(* Logix 5000 project; controller PRU vendor 1 type 14 code 107 rev 20.13; software revision 20.01; part 13 of 17 *)
(* tags used below, declared in another part *)
   AI0_CALCULATED : REAL;
   AI0_WF : DSi_WF50;
   AI10_CALCULATED : REAL;
   AI10_WF : DSi_WF50;
   AI11_CALCULATED : REAL;
   AI11_WF : DSi_WF50;
   AI12_CALCULATED : REAL;
   AI12_WF : DSi_WF50;
   AI13_CALCULATED : REAL;
   AI13_WF : DSi_WF50;
   AI14_CALCULATED : REAL;
   AI14_WF : DSi_WF50;
   AI15_CALCULATED : REAL;
   AI15_WF : DSi_WF50;
   AI16_CALCULATED : REAL;
   AI16_WF : DSi_WF50;
   AI1_CALCULATED : REAL;
   AI1_WF : DSi_WF50;
   AI2_CALCULATED : REAL;
   AI2_WF : DSi_WF50;
   AI3_CALCULATED : REAL;
   AI3_WF : DSi_WF50;
   AI4_CALCULATED : REAL;
   AI4_WF : DSi_WF50;
   AI5_CALCULATED : REAL;
   AI5_WF : DSi_WF50;
   AI6_CALCULATED : REAL;
   AI6_WF : DSi_WF50;
   AI7_CALCULATED : REAL;
   AI7_WF : DSi_WF50;
   AI8_CALCULATED : REAL;
   AI8_WF : DSi_WF50;
   AI9_CALCULATED : REAL;
   AI9_WF : DSi_WF50;
   AI_0 : AI_1769_IF4;
   AI_0_FILTERED : DINT;
   AI_1 : AI_1769_IF4;
   AI_10 : AI_1769_IF4;
   AI_10_FILTERED : REAL;
   AI_11 : AI_1769_IF4;
   AI_11_FILTERED : REAL;
   AI_12 : AI_1769_IF4;
   AI_12_FILTERED : REAL;
   AI_13 : AI_1769_IF4;
   AI_13_FILTERED : REAL;
   AI_14 : AI_1769_IF4;
   AI_14_FILTERED : REAL;
   AI_15 : AI_1769_IF4;
   AI_15_FILTERED : REAL;
   AI_16 : AI_1769_IF4;
   AI_16_DATA : REAL;
   AI_16_FILTERED : REAL;
   AI_1_FILTERED : REAL;
   AI_2 : AI_1769_IF4;
   AI_2_FILTERED : REAL;
   AI_3 : AI_1769_IF4;
   AI_3_FILTERED : REAL;
   AI_4 : AI_1769_IF4;
   AI_4_FILTERED : REAL;
   AI_5 : AI_1769_IF4;
   AI_5_FILTERED : REAL;
   AI_6 : AI_1769_IF4;
   AI_6_FILTERED : REAL;
   AI_7 : AI_1769_IF4;
   AI_7_FILTERED : REAL;
   AI_8 : AI_1769_IF4;
   AI_8_FILTERED : REAL;
   AI_9 : AI_1769_IF4;
   AI_9_FILTERED : REAL;
   CALC_SPARE_AO_CMD : REAL;
   CSS_CommsLoss_TMR : TIMER;
   CSS_CommsLossAlm : BOOL;
   CSS_CommsWarning_TMR : TIMER;
   CSS_CommsWarningAlm : BOOL;
   CSS_PLC_Seconds_Temp : DINT;
   CSS_Status_Data : PLCStatusData;
   DisableAllHeaters : BOOL;
   HMI_Ai0_FORCE : BOOL;
   HMI_Ai0_FORCE_VALUE : REAL;
   HMI_AI0_HI_SCALE : REAL;
   HMI_AI0_LO_SCALE : REAL;
   HMI_Ai10_FORCE : BOOL;
   HMI_Ai10_FORCE_VALUE : REAL;
   HMI_AI10_HI_SCALE : REAL;
   HMI_AI10_LO_SCALE : REAL;
   HMI_Ai11_FORCE : BOOL;
   HMI_Ai11_FORCE_VALUE : REAL;
   HMI_AI11_HI_SCALE : REAL;
   HMI_AI11_LO_SCALE : REAL;
   HMI_Ai12_FORCE : BOOL;
   HMI_Ai12_FORCE_VALUE : REAL;
   HMI_AI12_HI_SCALE : REAL;
   HMI_AI12_LO_SCALE : REAL;
   HMI_Ai13_FORCE : BOOL;
   HMI_Ai13_FORCE_VALUE : REAL;
   HMI_AI13_HI_SCALE : REAL;
   HMI_AI13_LO_SCALE : REAL;
   HMI_Ai14_FORCE : BOOL;
   HMI_Ai14_FORCE_VALUE : REAL;
   HMI_AI14_HI_SCALE : REAL;
   HMI_AI14_LO_SCALE : REAL;
   HMI_Ai15_FORCE : BOOL;
   HMI_Ai15_FORCE_VALUE : REAL;
   HMI_AI15_HI_SCALE : REAL;
   HMI_AI15_LO_SCALE : REAL;
   HMI_AI16_FORCE : BOOL;
   HMI_AI16_FORCE_VALUE : REAL;
   HMI_AI16_HI_SCALE : REAL;
   HMI_AI16_LO_SCALE : REAL;
   HMI_Ai1_FORCE : BOOL;
   HMI_Ai1_FORCE_VALUE : REAL;
   HMI_AI1_HI_SCALE : REAL;
   HMI_AI1_LO_SCALE : REAL;
   HMI_Ai2_FORCE : BOOL;
   HMI_Ai2_FORCE_VALUE : REAL;
   HMI_AI2_HI_SCALE : REAL;
   HMI_AI2_LO_SCALE : REAL;
   HMI_Ai3_FORCE : BOOL;
   HMI_Ai3_FORCE_VALUE : REAL;
   HMI_AI3_HI_SCALE : REAL;
   HMI_AI3_LO_SCALE : REAL;
   HMI_Ai4_FORCE : BOOL;
   HMI_Ai4_FORCE_VALUE : REAL;
   HMI_AI4_HI_SCALE : REAL;
   HMI_AI4_LO_SCALE : REAL;
   HMI_Ai5_FORCE : BOOL;
   HMI_Ai5_FORCE_VALUE : REAL;
   HMI_AI5_HI_SCALE : REAL;
   HMI_AI5_LO_SCALE : REAL;
   HMI_Ai6_FORCE : BOOL;
   HMI_Ai6_FORCE_VALUE : REAL;
   HMI_AI6_HI_SCALE : REAL;
   HMI_AI6_LO_SCALE : REAL;
   HMI_Ai7_FORCE : BOOL;
   HMI_Ai7_FORCE_VALUE : REAL;
   HMI_AI7_HI_SCALE : REAL;
   HMI_AI7_LO_SCALE : REAL;
   HMI_Ai8_FORCE : BOOL;
   HMI_Ai8_FORCE_VALUE : REAL;
   HMI_AI8_HI_SCALE : REAL;
   HMI_AI8_LO_SCALE : REAL;
   HMI_Ai9_FORCE : BOOL;
   HMI_Ai9_FORCE_VALUE : REAL;
   HMI_AI9_HI_SCALE : REAL;
   HMI_AI9_LO_SCALE : REAL;
   HMI_HTR1_FORCED : BOOL;
   HMI_HTR1_POWER_CMD : REAL;
   HMI_HTR2_FORCED : BOOL;
   HMI_HTR2_POWER_CMD : REAL;
   HMI_HTR3_FORCED : BOOL;
   HMI_HTR3_POWER_CMD : REAL;
   HMI_HTR4_FORCED : BOOL;
   HMI_HTR4_POWER_CMD : REAL;
   HMI_HTR5_FORCED : BOOL;
   HMI_HTR5_POWER_CMD : REAL;
   HMI_HTR6_FORCED : BOOL;
   HMI_HTR6_POWER_CMD : REAL;
   HMI_HTR7_FORCED : BOOL;
   HMI_HTR7_POWER_CMD : REAL;
   HMI_HTR8_FORCED : BOOL;
   HMI_HTR8_POWER_CMD : REAL;
   HMI_HTR9_FORCED : BOOL;
   HMI_HTR9_POWER_CMD : REAL;
   HMI_SPARE_AO_CMD : REAL;
   HMI_SPARE_AO_FORCED : BOOL;
   HTR1_POWER_CMD : REAL;
   HTR2_POWER_CMD : REAL;
   HTR3_POWER_CMD : REAL;
   HTR4_POWER_CMD : REAL;
   HTR5_POWER_CMD : REAL;
   HTR6_POWER_CMD : REAL;
   HTR7_POWER_CMD : REAL;
   HTR8_POWER_CMD : REAL;
   HTR9_POWER_CMD : REAL;
   Major : DINT;
   Minor : DINT;
   Revision : DINT;
   SPARE_AO_CMD : REAL;
   TOTE_WEIGHT : REAL;
   UTL_Status_Data : PLCStatusData;
   Z1_AMPS_TEMP : REAL;
   Z1_L1_AMPS : REAL;
   Z1_L2_AMPS : REAL;
   Z1_L3_AMPS : REAL;
   Z1L1_Tot : EnergyTot;
   Z1L2_Tot : EnergyTot;
   Z1L3_Tot : EnergyTot;
   Z2_AMPS_TEMP : REAL;
   Z2_L1_AMPS : REAL;
   Z2_L2_AMPS : REAL;
   Z2_L3_AMPS : REAL;
   Z2L1_Tot : EnergyTot;
   Z2L2_Tot : EnergyTot;
   Z2L3_Tot : EnergyTot;
   Z3_AMPS_TEMP : REAL;
   Z3_L1_AMPS : REAL;
   Z3_L2_AMPS : REAL;
   Z3_L3_AMPS : REAL;
   Z3L1_Tot : EnergyTot;
   Z3L2_Tot : EnergyTot;
   Z3L3_Tot : EnergyTot;
   Z4_L1_AMPS : REAL;
   Z4L1_Tot : EnergyTot;
   Z5_L2_AMPS : REAL;
   Z5L2_Tot : EnergyTot;
   Z6_L3_AMPS : REAL;
   Z6L3_Tot : EnergyTot;
   Z7_L1_AMPS : REAL;
   Z7L1_Tot : EnergyTot;
   Z8_L2_AMPS : REAL;
   Z8L2_Tot : EnergyTot;
   Z9_L3_AMPS : REAL;
   Z9L3_Tot : EnergyTot;
   ZONE_1_AMPS : DINT;
   ZONE_1_POWER_CMD : REAL;
   ZONE_2_AMPS : DINT;
   ZONE_2_POWER_CMD : REAL;
   ZONE_3_AMPS : DINT;
   ZONE_3_POWER_CMD : REAL;
   ZONE_4_AMPS : DINT;
   ZONE_4_POWER_CMD : REAL;
   ZONE_5_AMPS : DINT;
   ZONE_5_POWER_CMD : REAL;
   ZONE_6_AMPS : DINT;
   ZONE_6_POWER_CMD : REAL;
   ZONE_7_AMPS : DINT;
   ZONE_7_POWER_CMD : REAL;
   ZONE_8_AMPS : DINT;
   ZONE_8_POWER_CMD : REAL;
   ZONE_9_AMPS : DINT;
   ZONE_9_POWER_CMD : REAL;
(* MainProgram, continued *)

ROUTINE G04_MAP_ANALOG_INPUTS   (* ladder *)
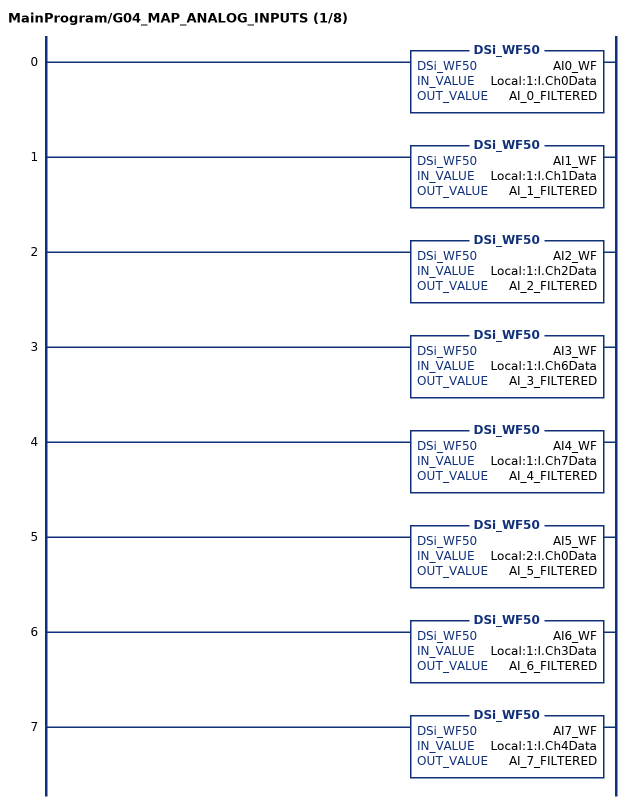
   0: DSi_WF50(AI0_WF,Local:1:I.Ch0Data,AI_0_FILTERED);
   1: DSi_WF50(AI1_WF,Local:1:I.Ch1Data,AI_1_FILTERED);
   2: DSi_WF50(AI2_WF,Local:1:I.Ch2Data,AI_2_FILTERED);
   3: DSi_WF50(AI3_WF,Local:1:I.Ch6Data,AI_3_FILTERED);
   4: DSi_WF50(AI4_WF,Local:1:I.Ch7Data,AI_4_FILTERED);
   5: DSi_WF50(AI5_WF,Local:2:I.Ch0Data,AI_5_FILTERED);
   6: DSi_WF50(AI6_WF,Local:1:I.Ch3Data,AI_6_FILTERED);
   7: DSi_WF50(AI7_WF,Local:1:I.Ch4Data,AI_7_FILTERED);
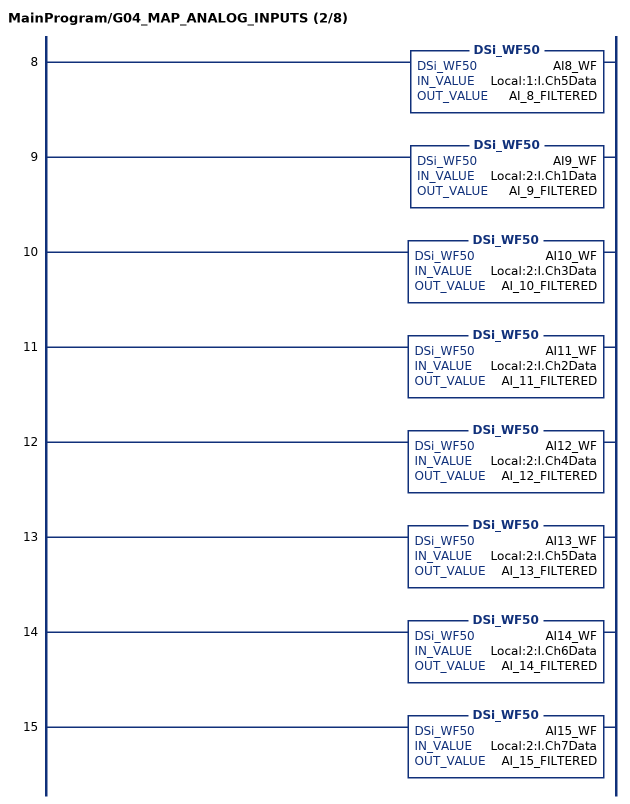
   8: DSi_WF50(AI8_WF,Local:1:I.Ch5Data,AI_8_FILTERED);
   9: DSi_WF50(AI9_WF,Local:2:I.Ch1Data,AI_9_FILTERED);
   10: DSi_WF50(AI10_WF,Local:2:I.Ch3Data,AI_10_FILTERED);
   11: DSi_WF50(AI11_WF,Local:2:I.Ch2Data,AI_11_FILTERED);
   12: DSi_WF50(AI12_WF,Local:2:I.Ch4Data,AI_12_FILTERED);
   13: DSi_WF50(AI13_WF,Local:2:I.Ch5Data,AI_13_FILTERED);
   14: DSi_WF50(AI14_WF,Local:2:I.Ch6Data,AI_14_FILTERED);
   15: DSi_WF50(AI15_WF,Local:2:I.Ch7Data,AI_15_FILTERED);
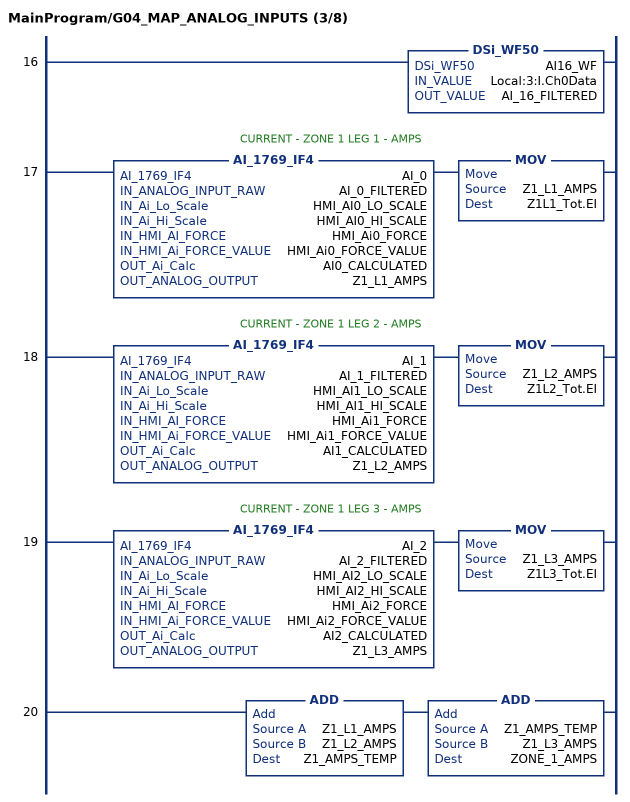
   16: DSi_WF50(AI16_WF,Local:3:I.Ch0Data,AI_16_FILTERED);
   // CURRENT - ZONE 1 LEG 1 - AMPS
   17: AI_1769_IF4(AI_0,AI_0_FILTERED,HMI_AI0_LO_SCALE,HMI_AI0_HI_SCALE,HMI_Ai0_FORCE,HMI_Ai0_FORCE_VALUE,AI0_CALCULATED,Z1_L1_AMPS)MOV(Z1_L1_AMPS,Z1L1_Tot.EI);
   // CURRENT - ZONE 1 LEG 2 - AMPS
   18: AI_1769_IF4(AI_1,AI_1_FILTERED,HMI_AI1_LO_SCALE,HMI_AI1_HI_SCALE,HMI_Ai1_FORCE,HMI_Ai1_FORCE_VALUE,AI1_CALCULATED,Z1_L2_AMPS)MOV(Z1_L2_AMPS,Z1L2_Tot.EI);
   // CURRENT - ZONE 1 LEG 3 - AMPS
   19: AI_1769_IF4(AI_2,AI_2_FILTERED,HMI_AI2_LO_SCALE,HMI_AI2_HI_SCALE,HMI_Ai2_FORCE,HMI_Ai2_FORCE_VALUE,AI2_CALCULATED,Z1_L3_AMPS)MOV(Z1_L3_AMPS,Z1L3_Tot.EI);
   20: ADD(Z1_L1_AMPS,Z1_L2_AMPS,Z1_AMPS_TEMP)ADD(Z1_AMPS_TEMP,Z1_L3_AMPS,ZONE_1_AMPS);
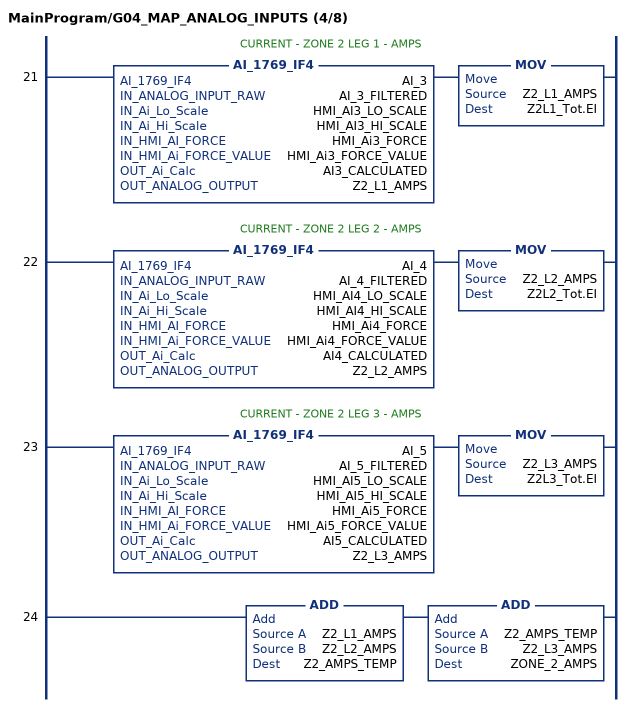
   // CURRENT - ZONE 2 LEG 1 - AMPS
   21: AI_1769_IF4(AI_3,AI_3_FILTERED,HMI_AI3_LO_SCALE,HMI_AI3_HI_SCALE,HMI_Ai3_FORCE,HMI_Ai3_FORCE_VALUE,AI3_CALCULATED,Z2_L1_AMPS)MOV(Z2_L1_AMPS,Z2L1_Tot.EI);
   // CURRENT - ZONE 2 LEG 2 - AMPS
   22: AI_1769_IF4(AI_4,AI_4_FILTERED,HMI_AI4_LO_SCALE,HMI_AI4_HI_SCALE,HMI_Ai4_FORCE,HMI_Ai4_FORCE_VALUE,AI4_CALCULATED,Z2_L2_AMPS)MOV(Z2_L2_AMPS,Z2L2_Tot.EI);
   // CURRENT - ZONE 2 LEG 3 - AMPS
   23: AI_1769_IF4(AI_5,AI_5_FILTERED,HMI_AI5_LO_SCALE,HMI_AI5_HI_SCALE,HMI_Ai5_FORCE,HMI_Ai5_FORCE_VALUE,AI5_CALCULATED,Z2_L3_AMPS)MOV(Z2_L3_AMPS,Z2L3_Tot.EI);
   24: ADD(Z2_L1_AMPS,Z2_L2_AMPS,Z2_AMPS_TEMP)ADD(Z2_AMPS_TEMP,Z2_L3_AMPS,ZONE_2_AMPS);
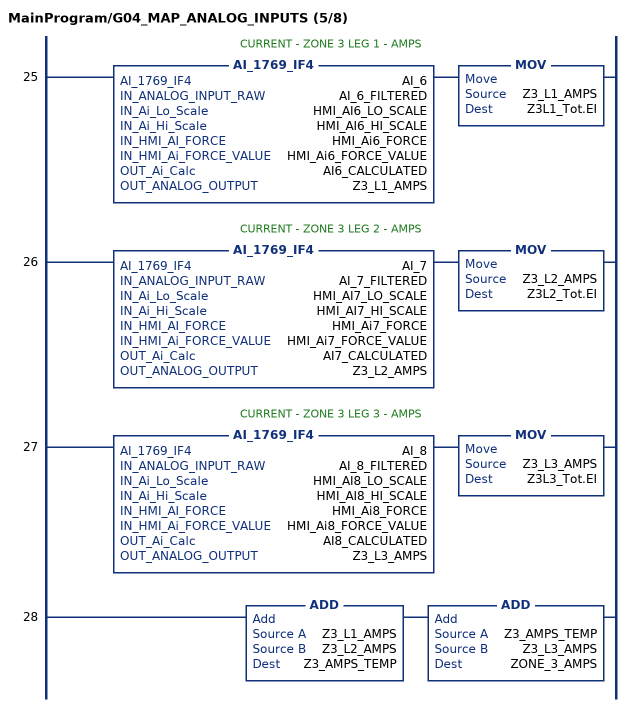
   // CURRENT - ZONE 3 LEG 1 - AMPS
   25: AI_1769_IF4(AI_6,AI_6_FILTERED,HMI_AI6_LO_SCALE,HMI_AI6_HI_SCALE,HMI_Ai6_FORCE,HMI_Ai6_FORCE_VALUE,AI6_CALCULATED,Z3_L1_AMPS)MOV(Z3_L1_AMPS,Z3L1_Tot.EI);
   // CURRENT - ZONE 3 LEG 2 - AMPS
   26: AI_1769_IF4(AI_7,AI_7_FILTERED,HMI_AI7_LO_SCALE,HMI_AI7_HI_SCALE,HMI_Ai7_FORCE,HMI_Ai7_FORCE_VALUE,AI7_CALCULATED,Z3_L2_AMPS)MOV(Z3_L2_AMPS,Z3L2_Tot.EI);
   // CURRENT - ZONE 3 LEG 3 - AMPS
   27: AI_1769_IF4(AI_8,AI_8_FILTERED,HMI_AI8_LO_SCALE,HMI_AI8_HI_SCALE,HMI_Ai8_FORCE,HMI_Ai8_FORCE_VALUE,AI8_CALCULATED,Z3_L3_AMPS)MOV(Z3_L3_AMPS,Z3L3_Tot.EI);
   28: ADD(Z3_L1_AMPS,Z3_L2_AMPS,Z3_AMPS_TEMP)ADD(Z3_AMPS_TEMP,Z3_L3_AMPS,ZONE_3_AMPS);
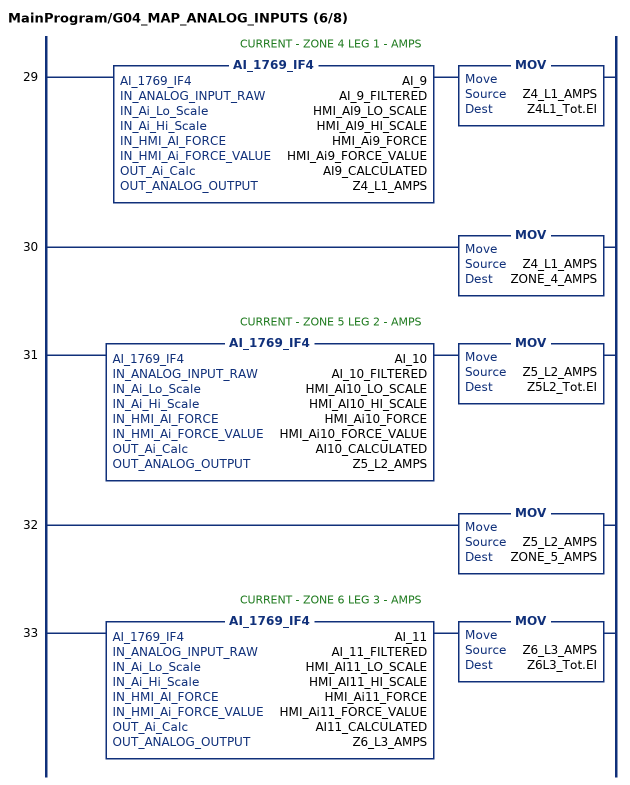
   // CURRENT - ZONE 4 LEG 1 - AMPS
   29: AI_1769_IF4(AI_9,AI_9_FILTERED,HMI_AI9_LO_SCALE,HMI_AI9_HI_SCALE,HMI_Ai9_FORCE,HMI_Ai9_FORCE_VALUE,AI9_CALCULATED,Z4_L1_AMPS)MOV(Z4_L1_AMPS,Z4L1_Tot.EI);
   30: MOV(Z4_L1_AMPS,ZONE_4_AMPS);
   // CURRENT - ZONE 5 LEG 2 - AMPS
   31: AI_1769_IF4(AI_10,AI_10_FILTERED,HMI_AI10_LO_SCALE,HMI_AI10_HI_SCALE,HMI_Ai10_FORCE,HMI_Ai10_FORCE_VALUE,AI10_CALCULATED,Z5_L2_AMPS)MOV(Z5_L2_AMPS,Z5L2_Tot.EI);
   32: MOV(Z5_L2_AMPS,ZONE_5_AMPS);
   // CURRENT - ZONE 6 LEG 3 - AMPS
   33: AI_1769_IF4(AI_11,AI_11_FILTERED,HMI_AI11_LO_SCALE,HMI_AI11_HI_SCALE,HMI_Ai11_FORCE,HMI_Ai11_FORCE_VALUE,AI11_CALCULATED,Z6_L3_AMPS)MOV(Z6_L3_AMPS,Z6L3_Tot.EI);
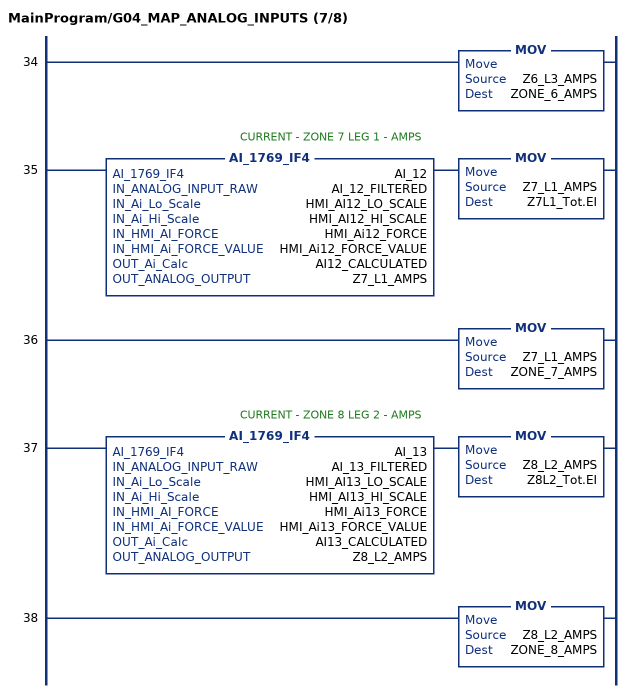
   34: MOV(Z6_L3_AMPS,ZONE_6_AMPS);
   // CURRENT - ZONE 7 LEG 1 - AMPS
   35: AI_1769_IF4(AI_12,AI_12_FILTERED,HMI_AI12_LO_SCALE,HMI_AI12_HI_SCALE,HMI_Ai12_FORCE,HMI_Ai12_FORCE_VALUE,AI12_CALCULATED,Z7_L1_AMPS)MOV(Z7_L1_AMPS,Z7L1_Tot.EI);
   36: MOV(Z7_L1_AMPS,ZONE_7_AMPS);
   // CURRENT - ZONE 8 LEG 2 - AMPS
   37: AI_1769_IF4(AI_13,AI_13_FILTERED,HMI_AI13_LO_SCALE,HMI_AI13_HI_SCALE,HMI_Ai13_FORCE,HMI_Ai13_FORCE_VALUE,AI13_CALCULATED,Z8_L2_AMPS)MOV(Z8_L2_AMPS,Z8L2_Tot.EI);
   38: MOV(Z8_L2_AMPS,ZONE_8_AMPS);
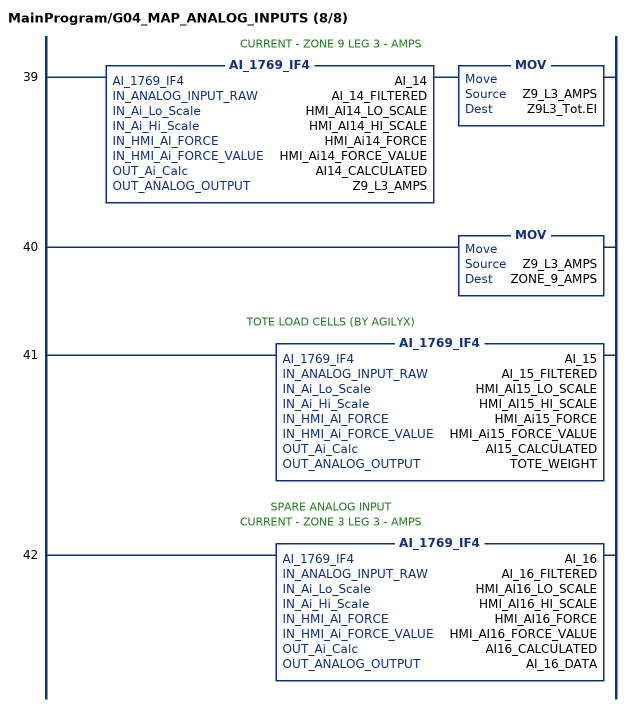
   // CURRENT - ZONE 9 LEG 3 - AMPS
   39: AI_1769_IF4(AI_14,AI_14_FILTERED,HMI_AI14_LO_SCALE,HMI_AI14_HI_SCALE,HMI_Ai14_FORCE,HMI_Ai14_FORCE_VALUE,AI14_CALCULATED,Z9_L3_AMPS)MOV(Z9_L3_AMPS,Z9L3_Tot.EI);
   40: MOV(Z9_L3_AMPS,ZONE_9_AMPS);
   // TOTE LOAD CELLS (BY AGILYX)
   41: AI_1769_IF4(AI_15,AI_15_FILTERED,HMI_AI15_LO_SCALE,HMI_AI15_HI_SCALE,HMI_Ai15_FORCE,HMI_Ai15_FORCE_VALUE,AI15_CALCULATED,TOTE_WEIGHT);
   // SPARE ANALOG INPUT
   // CURRENT - ZONE 3 LEG 3 - AMPS
   42: AI_1769_IF4(AI_16,AI_16_FILTERED,HMI_AI16_LO_SCALE,HMI_AI16_HI_SCALE,HMI_AI16_FORCE,HMI_AI16_FORCE_VALUE,AI16_CALCULATED,AI_16_DATA);
END_ROUTINE

ROUTINE G05_MAP_ANALOG_OUTPUTS   (* ladder *)
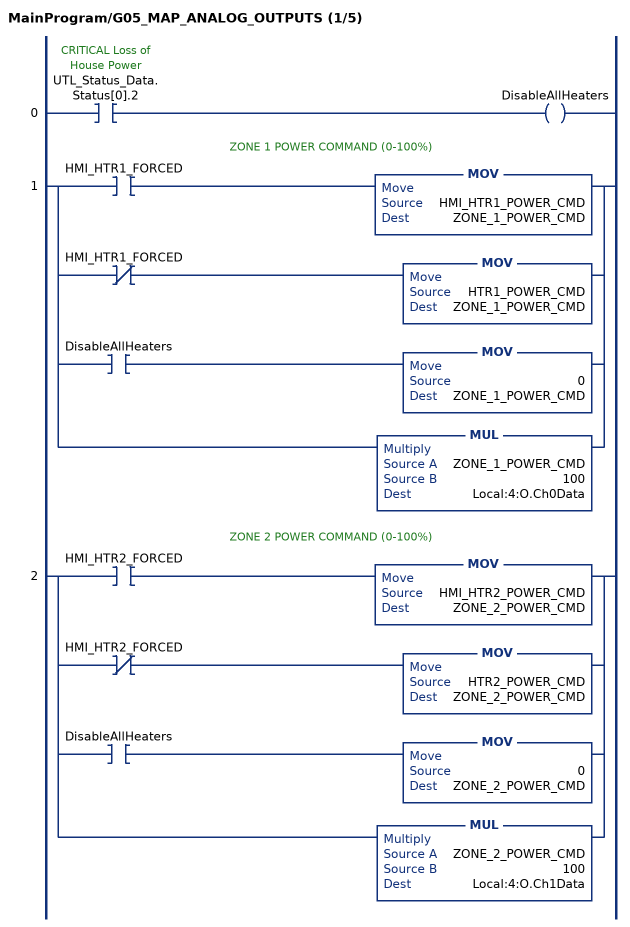
   0: XIC(UTL_Status_Data.Status[0].2)OTE(DisableAllHeaters);
   // ZONE 1 POWER COMMAND (0-100%)
   1: [XIC(HMI_HTR1_FORCED) MOV(HMI_HTR1_POWER_CMD,ZONE_1_POWER_CMD) ,XIO(HMI_HTR1_FORCED) MOV(HTR1_POWER_CMD,ZONE_1_POWER_CMD) ,XIC(DisableAllHeaters) MOV(0,ZONE_1_POWER_CMD) ,MUL(ZONE_1_POWER_CMD,100,Local:4:O.Ch0Data) ];
   // ZONE 2 POWER COMMAND (0-100%)
   2: [XIC(HMI_HTR2_FORCED) MOV(HMI_HTR2_POWER_CMD,ZONE_2_POWER_CMD) ,XIO(HMI_HTR2_FORCED) MOV(HTR2_POWER_CMD,ZONE_2_POWER_CMD) ,XIC(DisableAllHeaters) MOV(0,ZONE_2_POWER_CMD) ,MUL(ZONE_2_POWER_CMD,100,Local:4:O.Ch1Data) ];
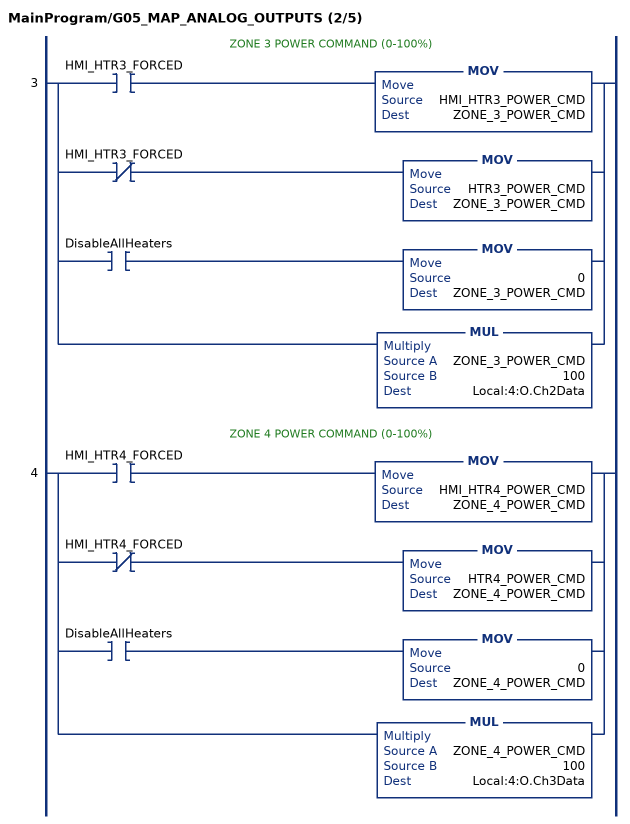
   // ZONE 3 POWER COMMAND (0-100%)
   3: [XIC(HMI_HTR3_FORCED) MOV(HMI_HTR3_POWER_CMD,ZONE_3_POWER_CMD) ,XIO(HMI_HTR3_FORCED) MOV(HTR3_POWER_CMD,ZONE_3_POWER_CMD) ,XIC(DisableAllHeaters) MOV(0,ZONE_3_POWER_CMD) ,MUL(ZONE_3_POWER_CMD,100,Local:4:O.Ch2Data) ];
   // ZONE 4 POWER COMMAND (0-100%)
   4: [XIC(HMI_HTR4_FORCED) MOV(HMI_HTR4_POWER_CMD,ZONE_4_POWER_CMD) ,XIO(HMI_HTR4_FORCED) MOV(HTR4_POWER_CMD,ZONE_4_POWER_CMD) ,XIC(DisableAllHeaters) MOV(0,ZONE_4_POWER_CMD) ,MUL(ZONE_4_POWER_CMD,100,Local:4:O.Ch3Data) ];
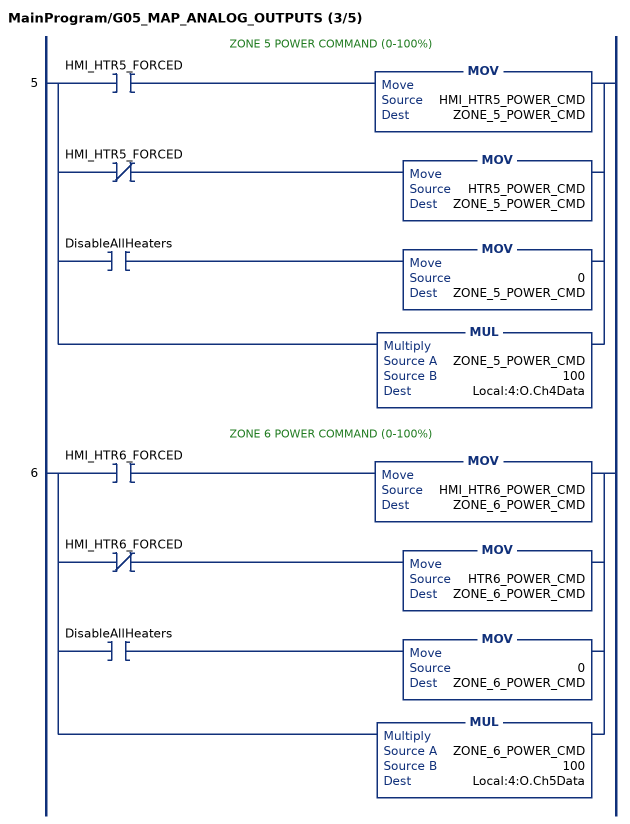
   // ZONE 5 POWER COMMAND (0-100%)
   5: [XIC(HMI_HTR5_FORCED) MOV(HMI_HTR5_POWER_CMD,ZONE_5_POWER_CMD) ,XIO(HMI_HTR5_FORCED) MOV(HTR5_POWER_CMD,ZONE_5_POWER_CMD) ,XIC(DisableAllHeaters) MOV(0,ZONE_5_POWER_CMD) ,MUL(ZONE_5_POWER_CMD,100,Local:4:O.Ch4Data) ];
   // ZONE 6 POWER COMMAND (0-100%)
   6: [XIC(HMI_HTR6_FORCED) MOV(HMI_HTR6_POWER_CMD,ZONE_6_POWER_CMD) ,XIO(HMI_HTR6_FORCED) MOV(HTR6_POWER_CMD,ZONE_6_POWER_CMD) ,XIC(DisableAllHeaters) MOV(0,ZONE_6_POWER_CMD) ,MUL(ZONE_6_POWER_CMD,100,Local:4:O.Ch5Data) ];
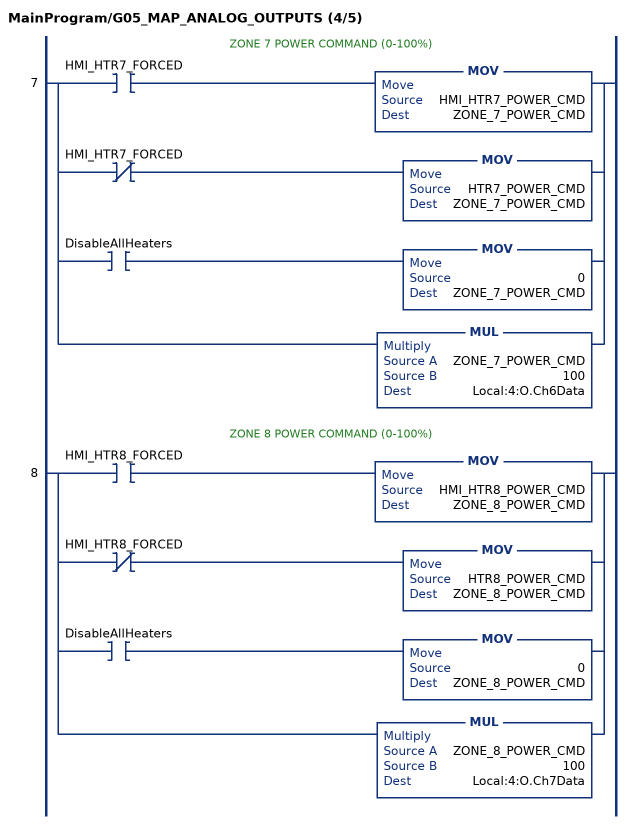
   // ZONE 7 POWER COMMAND (0-100%)
   7: [XIC(HMI_HTR7_FORCED) MOV(HMI_HTR7_POWER_CMD,ZONE_7_POWER_CMD) ,XIO(HMI_HTR7_FORCED) MOV(HTR7_POWER_CMD,ZONE_7_POWER_CMD) ,XIC(DisableAllHeaters) MOV(0,ZONE_7_POWER_CMD) ,MUL(ZONE_7_POWER_CMD,100,Local:4:O.Ch6Data) ];
   // ZONE 8 POWER COMMAND (0-100%)
   8: [XIC(HMI_HTR8_FORCED) MOV(HMI_HTR8_POWER_CMD,ZONE_8_POWER_CMD) ,XIO(HMI_HTR8_FORCED) MOV(HTR8_POWER_CMD,ZONE_8_POWER_CMD) ,XIC(DisableAllHeaters) MOV(0,ZONE_8_POWER_CMD) ,MUL(ZONE_8_POWER_CMD,100,Local:4:O.Ch7Data) ];
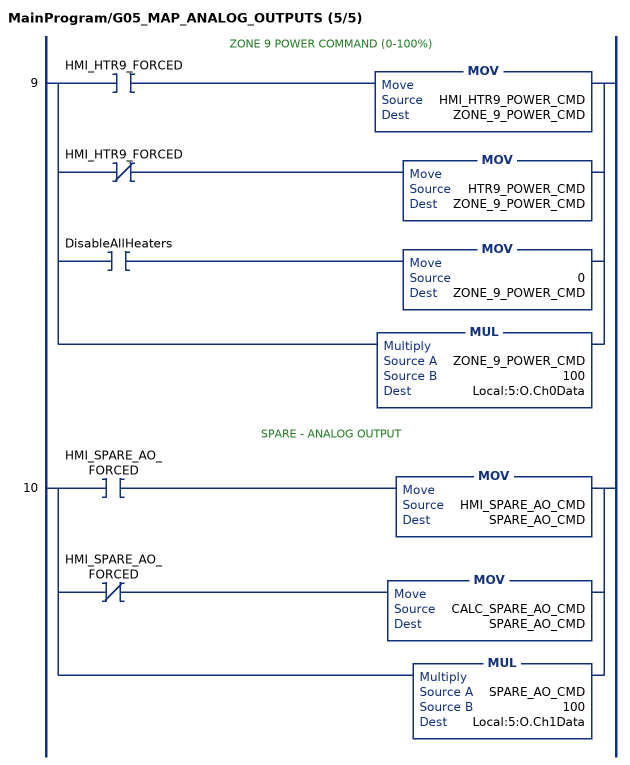
   // ZONE 9 POWER COMMAND (0-100%)
   9: [XIC(HMI_HTR9_FORCED) MOV(HMI_HTR9_POWER_CMD,ZONE_9_POWER_CMD) ,XIO(HMI_HTR9_FORCED) MOV(HTR9_POWER_CMD,ZONE_9_POWER_CMD) ,XIC(DisableAllHeaters) MOV(0,ZONE_9_POWER_CMD) ,MUL(ZONE_9_POWER_CMD,100,Local:5:O.Ch0Data) ];
   // SPARE - ANALOG OUTPUT
   10: [XIC(HMI_SPARE_AO_FORCED) MOV(HMI_SPARE_AO_CMD,SPARE_AO_CMD) ,XIO(HMI_SPARE_AO_FORCED) MOV(CALC_SPARE_AO_CMD,SPARE_AO_CMD) ,MUL(SPARE_AO_CMD,100,Local:5:O.Ch1Data) ];
END_ROUTINE

ROUTINE MainRoutine   (* ladder *)
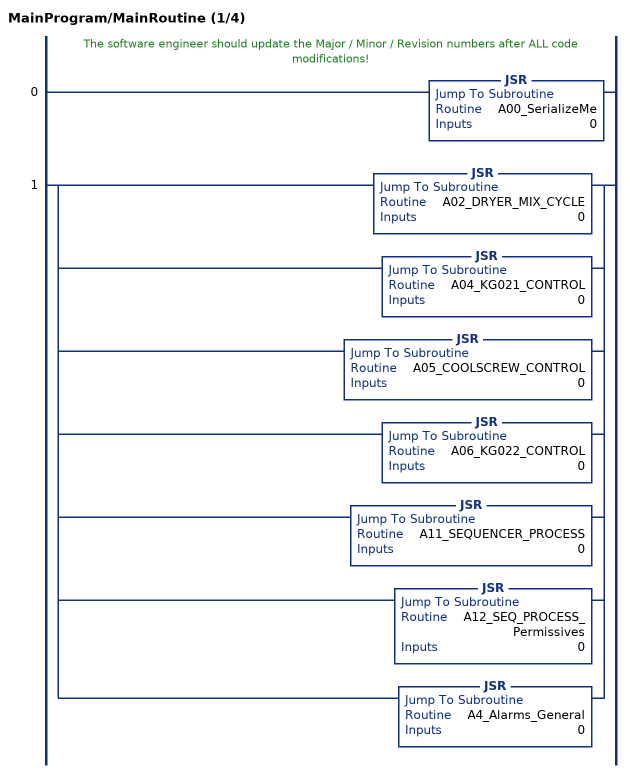
   // The software engineer should update the Major / Minor / Revision numbers after ALL code modifications!
   0: JSR(A00_SerializeMe,0);
   1: [JSR(A02_DRYER_MIX_CYCLE,0) ,JSR(A04_KG021_CONTROL,0) ,JSR(A05_COOLSCREW_CONTROL,0) ,JSR(A06_KG022_CONTROL,0) ,JSR(A11_SEQUENCER_PROCESS,0) ,JSR(A12_SEQ_PROCESS_Permissives,0) ,JSR(A4_Alarms_General,0) ];
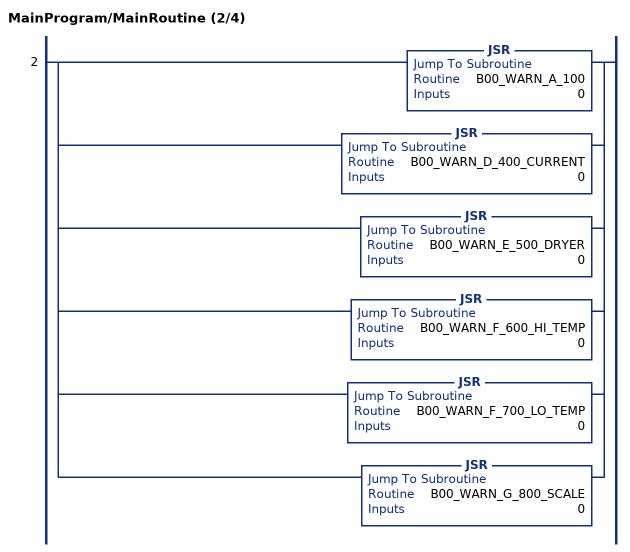
   2: [JSR(B00_WARN_A_100,0) ,JSR(B00_WARN_D_400_CURRENT,0) ,JSR(B00_WARN_E_500_DRYER,0) ,JSR(B00_WARN_F_600_HI_TEMP,0) ,JSR(B00_WARN_F_700_LO_TEMP,0) ,JSR(B00_WARN_G_800_SCALE,0) ];
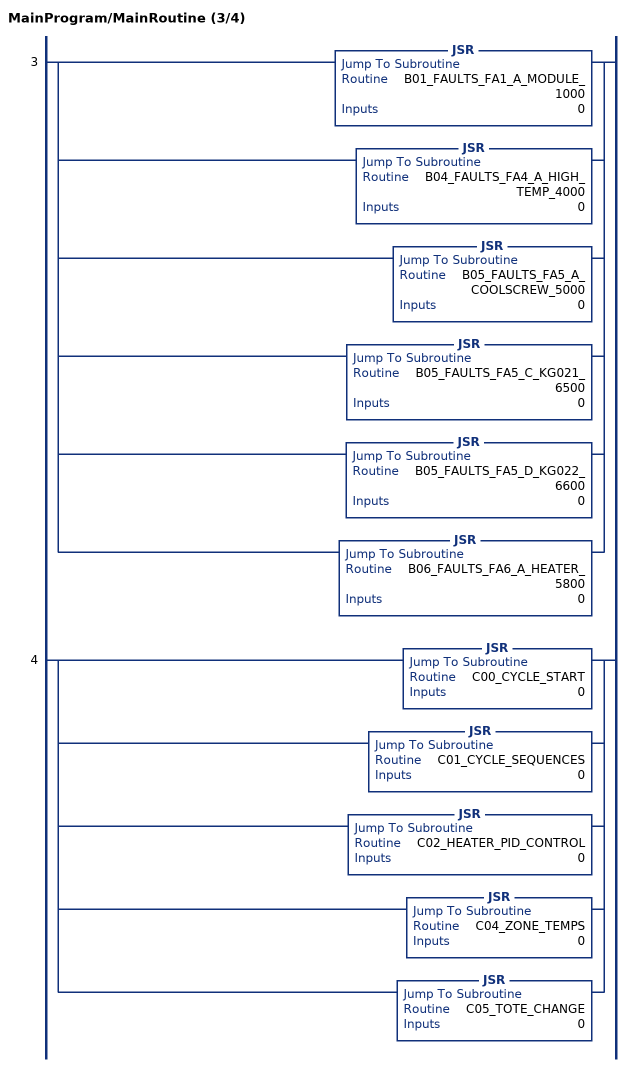
   3: [JSR(B01_FAULTS_FA1_A_MODULE_1000,0) ,JSR(B04_FAULTS_FA4_A_HIGH_TEMP_4000,0) ,JSR(B05_FAULTS_FA5_A_COOLSCREW_5000,0) ,JSR(B05_FAULTS_FA5_C_KG021_6500,0) ,JSR(B05_FAULTS_FA5_D_KG022_6600,0) ,JSR(B06_FAULTS_FA6_A_HEATER_5800,0) ];
   4: [JSR(C00_CYCLE_START,0) ,JSR(C01_CYCLE_SEQUENCES,0) ,JSR(C02_HEATER_PID_CONTROL,0) ,JSR(C04_ZONE_TEMPS,0) ,JSR(C05_TOTE_CHANGE,0) ];
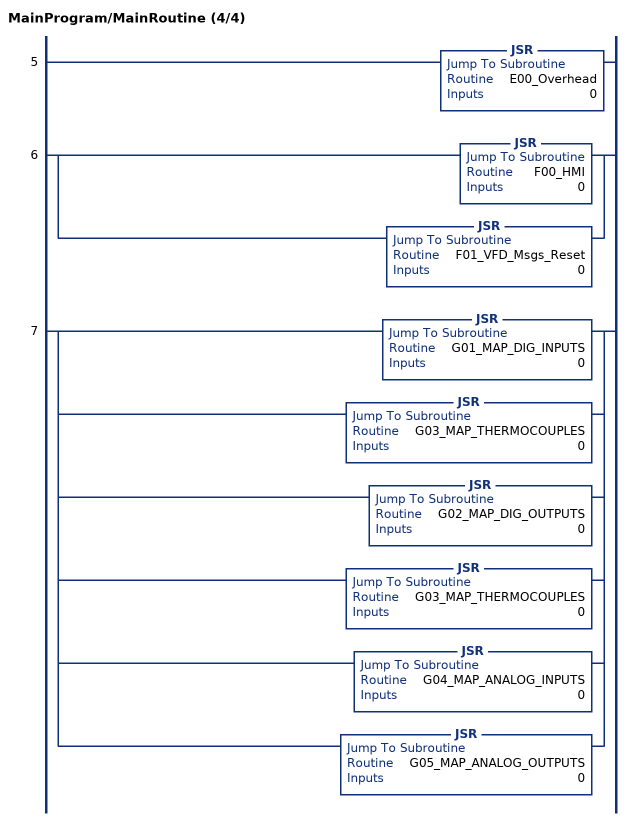
   5: JSR(E00_Overhead,0);
   6: [JSR(F00_HMI,0) ,JSR(F01_VFD_Msgs_Reset,0) ];
   7: [JSR(G01_MAP_DIG_INPUTS,0) ,JSR(G03_MAP_THERMOCOUPLES,0) ,JSR(G02_MAP_DIG_OUTPUTS,0) ,JSR(G03_MAP_THERMOCOUPLES,0) ,JSR(G04_MAP_ANALOG_INPUTS,0) ,JSR(G05_MAP_ANALOG_OUTPUTS,0) ];
END_ROUTINE
END_PROGRAM

PROGRAM MSG   (* main routine MSG *)

ROUTINE CSS_MSG   (* ladder *)
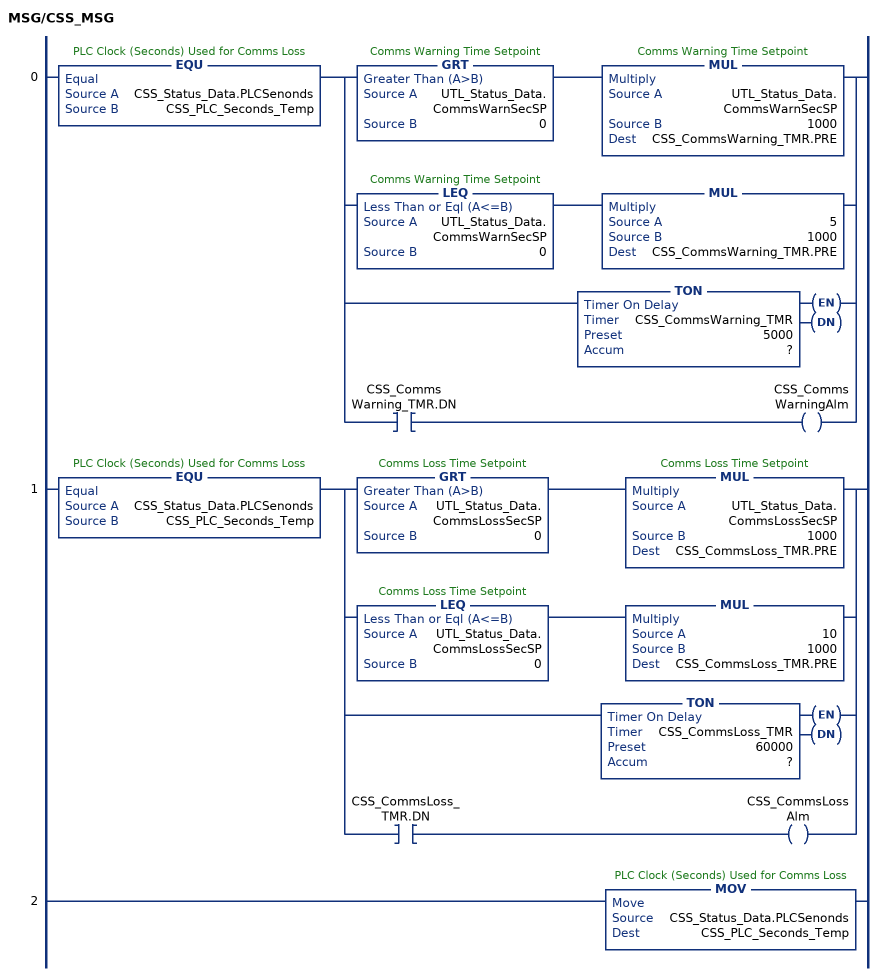
   0: EQU(CSS_Status_Data.PLCSenonds,CSS_PLC_Seconds_Temp)[GRT(UTL_Status_Data.CommsWarnSecSP,0) MUL(UTL_Status_Data.CommsWarnSecSP,1000,CSS_CommsWarning_TMR.PRE) ,LEQ(UTL_Status_Data.CommsWarnSecSP,0) MUL(5,1000,CSS_CommsWarning_TMR.PRE) ,TON(CSS_CommsWarning_TMR,?,?) ,XIC(CSS_CommsWarning_TMR.DN) OTE(CSS_CommsWarningAlm) ];
   1: EQU(CSS_Status_Data.PLCSenonds,CSS_PLC_Seconds_Temp)[GRT(UTL_Status_Data.CommsLossSecSP,0) MUL(UTL_Status_Data.CommsLossSecSP,1000,CSS_CommsLoss_TMR.PRE) ,LEQ(UTL_Status_Data.CommsLossSecSP,0) MUL(10,1000,CSS_CommsLoss_TMR.PRE) ,TON(CSS_CommsLoss_TMR,?,?) ,XIC(CSS_CommsLoss_TMR.DN) OTE(CSS_CommsLossAlm) ];
   2: MOV(CSS_Status_Data.PLCSenonds,CSS_PLC_Seconds_Temp);
END_ROUTINE
